(* PLC project Programme MGS_2-07_refactorJOY.project, CODESYS CODESYS V3.5 SP19 Patch 1 *)
(* stored: creationDateTime 2026-06-29T23:37:41.1568952, modificationDateTime 2026-06-29T22:49:33.424 *)

{attribute 'object_name' := 'diagETHERCAT'}
FUNCTION_BLOCK diagETHERCAT
  VAR_INPUT
    Enable : BOOL;  (* Active la surveillance *)
    Reset : BOOL;  (* Acquittement des défauts *)
    WcState : BOOL;  (* Working Counter (FALSE = Trame valide/En ligne) *)
    SlaveState : WORD;  (* État interne esclave (8 = OP / Operational) *)
  END_VAR
  VAR_OUTPUT
    Ready : BOOL;  (* Bloc actif *)
    Online : BOOL;  (* Esclave présent et répond *)
    Operational : BOOL;  (* Esclave en mode OP (données valides) *)
    Error : BOOL;  (* Défaut actif *)
    ErrorId : WORD;  (* Code d'erreur *)
  END_VAR

            // 🛑 1. GATE DE SÉCURITÉ
IF NOT Enable THEN
    Ready := FALSE;
    Online := FALSE;
    Operational := FALSE;
    Error := FALSE;
    ErrorId := 16#0000;
    RETURN;
END_IF;

Ready := TRUE;

// 🔑 2. RESET DÉFAUT
IF Reset AND Error THEN
    Error := FALSE;
    ErrorId := 16#0000;
END_IF;

// 🔍 3. DIAGNOSTIC ETHERCAT
// WcState à FALSE signifie que le maître communique physiquement avec le nœud
Online := NOT WcState; 

// L'état 8 en EtherCAT correspond à l'état "Operational" (échanges cycliques actifs)
Operational := Online AND (SlaveState = 8);

// ⚠️ 4. GESTION DES ERREURS
IF NOT Online THEN
    Error := TRUE;
    ErrorId := 16#0010; // Code : Perte de communication physique
ELSIF NOT Operational THEN
    Error := TRUE;
    ErrorId := 16#0011; // Code : Esclave hors mode Operational (Pre-Op, Safe-Op, etc.)
END_IF;
          
END_FUNCTION_BLOCK
